(* IEC 61131-3 sources: Industry-PLC-LLM/data/PLCBEAD_repo/PLCBEAD_PLCEmbed-main/PLC-BEAD/Source/GEB/DAY_OF_YEAR, 1 file *)

(* ---- DAY_OF_YEAR.ST ---- *)
FUNCTION DAY_OF_YEAR:INT
	VAR_INPUT
		IDATE :	DATE;
	END_VAR

	DAY_OF_YEAR  := UDINT_TO_INT((DATE_TO_UDINT(IDATE) / UDINT#86400) MOD UDINT#1461);
	IF DAY_OF_YEAR  > 729 THEN
		IF DAY_OF_YEAR  > 1095 THEN DAY_OF_YEAR  := DAY_OF_YEAR  - 1095; ELSE DAY_OF_YEAR  := DAY_OF_YEAR  - 729; END_IF;
	ELSIF DAY_OF_YEAR  > 364 THEN
		DAY_OF_YEAR  := DAY_OF_YEAR  - 364;
	ELSE
		DAY_OF_YEAR  := DAY_OF_YEAR  + 1;
	END_IF;
END_FUNCTION

PROGRAM program0
  VAR
    LocalVar0 : DATE;
	LocalOUT  : INT;
  END_VAR
  	LocalOUT := DAY_OF_YEAR(LocalVar0);
END_PROGRAM
